{attribute 'GeneratedUsingTerminal: EL2212-0000-0018'}
{attribute addProperty BoxType "EL2212-0000-0018"}
{attribute addProperty Id "StatusAT %I*Status_D9DC9C1B7"}
{attribute addProperty CRC "165496264"}
{attribute addProperty Size "7"}
TYPE DOX_Status_Channel_09DD45C8 :
STRUCT
	{attribute addProperty Name "Status"}
	Status AT %I* : Status_D9DC9C1B;
END_STRUCT
END_TYPE

(* stored: Version 1.2.0.0, ProductVersion 3.1.4024.9
   DUT DOX_Status_Channel_09DD45C8: Id {11b722ec-0198-40f8-9440-655b8a3e15b6} *)
